// Block: PPrgArchive19

DATA_BLOCK PPrgArchive19
VERSION : 0.1
   NON_RETAIN
   VAR
      PRG : Array[1801..1900] of PPrg_Data;
   END_VAR

BEGIN
   // No initialization required
END_DATA_BLOCK
